RoboDK station: ScaraExample.rdk

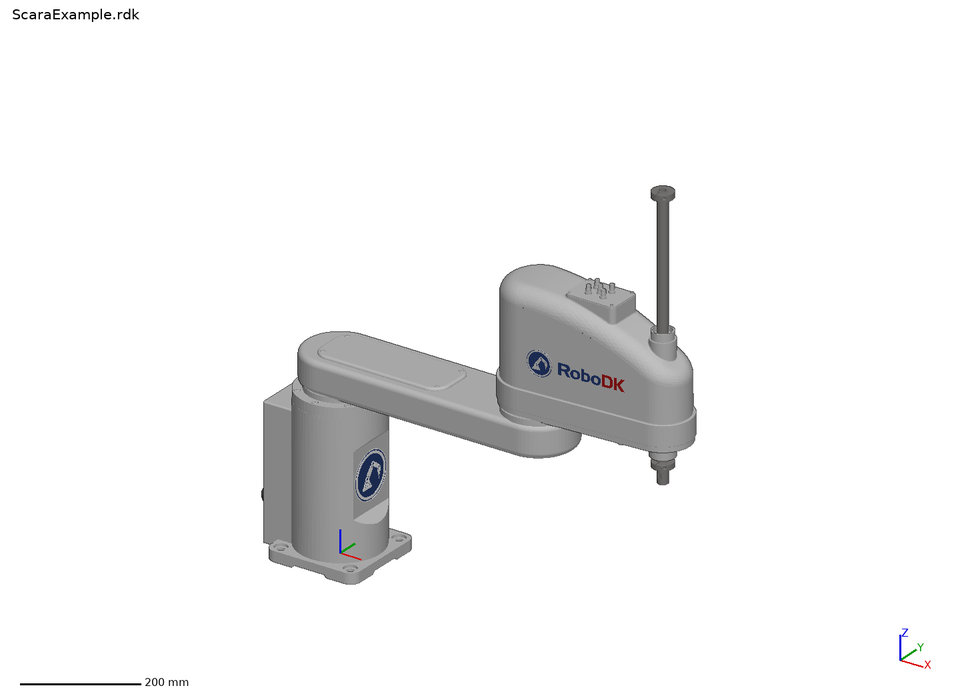
[picture v0: the station drawn from its stored meshes, robots at their saved joint values, targets as dots, program paths as lines]
Station ScaraExample (saved by RoboDK 6.0.0). Poses are relative to the parent item; angles as X-Y-Z fixed-axis rotations.
Station parameters (name, value as stored): LIN64
  - frame RoboDK RDK-SCARA-750 Base at (0, 0, 0) mm
    - robot RoboDK RDK-SCARA-750: 4 axes
        modified DH rows (alpha deg, a mm, theta deg, d mm): 0, 0, 0, 0; 0, 400, 0, 0; 0, 250, 0, 312 linear; 180, 0, 0, 0
        joint limits [-180, -150, -240, -360] to [180, 150, 0, 360]; home [0, 0, 0, 0]; saved at [0, 0, 0, 0]
  - Python program prog1 (listed below)

--- Python program prog1 ---
from robodk.robolink import Robolink, ITEM_TYPE_ROBOT
from robodk.robomath import transl, rotz

RDK = Robolink()

# Load your station
station_path = r"/home/KQ/Documents/Robotica/RoboDK/Stations/New Station (1).rdk"
RDK.AddFile(station_path)

# Pick the SCARA robot
robot = RDK.ItemUserPick("Seleccione el robot", ITEM_TYPE_ROBOT)
if not robot.Valid():
    raise Exception("No se seleccionó un robot válido")

# Points in mm (pick Z that is inside the SCARA's Z stroke)
puntos = [
    (200, 0,   200),
    (300, 0,   200),
    (300, 100, 200),
    (200, 100, 200),
]

# Keep a constant yaw (rotation around Z). For SCARA, this is typically fine.
yaw_deg = 0
yaw = yaw_deg * 3.1415926535 / 180.0

for x, y, z in puntos:
    pose = transl(x, y, z) * rotz(yaw)

    # Optional: check IK before moving (prevents crashing)
    jnts = robot.SolveIK(pose)
    if jnts is None or len(jnts) == 0:
        print(f"NOT reachable: {(x,y,z)}")
        continue

    print(f"Moving to: {(x,y,z)}")
    robot.MoveJ(pose)

# Return to first point
x0, y0, z0 = puntos[0]
robot.MoveJ(transl(x0, y0, z0) * rotz(yaw))

print("Programa finalizado.")
